(* Logix 5000 project; controller cal1615 1756-L62 rev 20.11; software revision 20.05; part 37 of 82 *)
(* tags used below, declared in another part *)
   FAULT : BOOL;   // Fault AFI
   p01_param_turret_dia_ft : REAL;
   p01r02 : routine;   // System Misc Control
   p01r09_pb_global_reset : BOOL;   // System Modes PB: Global Fault Reset
   p01r12_selected_line_speed : REAL;   // System Line Accel Decel Control Selected Line Speed
   p01r13_line_running : BOOL;   // System Line Start Sequence Line Running
   p01r13_line_slow_ramp : BOOL;   // System Line Start Sequence Start Line to Slow Speed
   p13r03_hz : SYS_SCP;   // Zone 3 Analog Inputs SCP Hz
   p20_acc_fill_time_sec : REAL;   // Letoff Accumulator Fill Time
   p20_acc_input_max : REAL;
   p20_acc_input_min : REAL;
   p20_acc_output_max : REAL;
   p20_acc_output_min : REAL;
   p20_ai_acc_pstn : REAL;   // Letoff Analog Input Accumulator Position
   p20_ai_lc01 : REAL;   // Letoff Analog Input Line Tension Load Cell Splicer
   p20_ai_letoff_dia : REAL;   // Letoff Analog Inputs Letoff Roll Diameter [in]
   p20_ai_lo_turret_amps : REAL;   // Letoff Inputs Letoff Turret VFD Amps
   p20_ai_lo_turret_hz : REAL;   // Letoff Inputs Letoff Turret VFD Hz
   p20_ai_lo_turret_speed : REAL;
   p20_ai_loa_speed : REAL;   // Letoff Inputs Letoff A VFD Surface Speed
   p20_ai_lob_speed : REAL;   // Letoff Inputs Letoff A Speed
   p20_di_acc_door_open : BOOL;
   p20_di_acc_empty : BOOL;   // Letoff Digital Input Letoff Accumulator Empty Position
   p20_di_acc_full : BOOL;   // Letoff Digital Input Letoff Accumulator Full Control Position
   p20_di_clutch_prs_ok : BOOL;   // Letoff Modes Accumulator Position Mode
   p20_di_lfr_jog_fwd : BOOL;   // Letoff Digital Input PB: Feedroll Jog Forward
   p20_di_lfr_jog_rev : BOOL;   // Letoff Digital Input PB: Feedroll Jog Reverse
   p20_di_lfr_nip_close : BOOL;   // Letoff Digital Input PB: Feedroll Nip Roll Close
   p20_di_lo_turret : acs800_di_normal;   // Letoff Letoff Turret VFD Drive Inputs
   p20_di_lo_turret_therm : BOOL;   // Letoff Input Letoff Turret Motor Temp Ok
   p20_di_loa_active : BOOL;   // Letoff Digital Input Letoff A Active
   p20_di_loa_brake : BOOL;   // Letoff Input Letoff A Brake Temperature Ok
   p20_di_loa_fwd_dir : BOOL;   // Letoff Digital Inputs PB: Letoff A Jog FWD
   p20_di_loa_jog : BOOL;   // Letoff Digital Inputs PB: Letoff A Jog REV
   p20_di_loa_start : BOOL;   // Letoff Digital Input PB: Letoff A Start
   p20_di_loa_stop : BOOL;   // Letoff Digital Input PB: Letoff A Stop Stop = 0
   p20_di_loa_temp : BOOL;   // Letoff Input Letoff A Motor Temperature Ok
   p20_di_lob_brake_thermostat : BOOL;   // Letoff Input Letoff B Brake Temperature OK
   p20_di_lob_fwd_dir : BOOL;   // Letoff Digital Inputs PB: Letoff B Jog FWD
   p20_di_lob_jog : BOOL;   // Letoff Digital Inputs PB: Letoff B Jog REV
   p20_di_lob_motor_thermostat : BOOL;   // Letoff Input Letoff B Motor Temperature Ok
   p20_di_lob_start : BOOL;   // Letoff Digital Input PB: Letoff B Start
   p20_di_lob_stop : BOOL;   // Letoff Digital Input PB: Letoff B Stop
   p20_di_lof_acc_fill : BOOL;   // Letoff Digital Input PB: Accumulator Fill
   p20_di_turret_fwd : BOOL;   // Letoff Digital Inputs PB: Turret FWD
   p20_di_turret_pos : BOOL;   // Letoff Digital Inputs PX: Turret in Position
   p20_di_turret_rev : BOOL;   // Letoff Digital Inputs PB: Turret REV
   p20_dia_input_max : REAL;
   p20_dia_input_min : REAL;
   p20_dia_output_max : REAL;
   p20_dia_output_min : REAL;
   p20_dint_to_hmi : DINT[16];   // Letoff Dint to HMI
   p20_lc_input_max : REAL;
   p20_lc_input_min : REAL;   // Letoff Analog Input
   p20_lc_output_max : REAL;
   p20_lc_output_min : REAL;
   p20_loa_ai_amps : REAL;   // Letoff Inputs Letoff A VFD Amps
   p20_loa_ai_hz : REAL;   // Letoff Inputs Letoff A Hz
   p20_loa_ai_rpm : REAL;
   p20_loa_ai_torque : REAL;
   p20_loa_footage_input_max : REAL;
   p20_loa_footage_input_min : REAL;
   p20_loa_footage_output_max : REAL;
   p20_loa_footage_output_min : REAL;
   p20_lob_ai_amps : REAL;   // Letoff Inputs Letoff B VFD Amps
   p20_lob_ai_hz : REAL;   // Letoff Inputs Letoff B VFD Hz
   p20_lob_ai_rpm : REAL;
   p20_lob_ai_torque : REAL;
   p20_lob_footage_input_max : REAL;
   p20_lob_footage_input_min : REAL;
   p20_lob_footage_output_max : REAL;
   p20_lob_footage_output_min : REAL;
   p20_param_lo_turret_gear_ratio : REAL;
   p20_param_loa_gear_ratio : REAL;
   p20_param_lob_gear_ratio : REAL;
   p20_vfd_di_loa : acs800_di_normal;   // Letoff A VFD Inputs
   p20_vfd_di_lob : acs800_di_normal;   // Letoff B VFD Inputs
   p20r01 : routine;   // Letoff Main
   p20r02 : routine;   // Letoff Misc Control
   p20r02_fault_exists : BOOL;
   p20r02_letoff_dia_ft : REAL;   // Letoff Misc Control Letoff Diameter [ft]
   p20r02_letoff_selection_dwell : TIMER;
   p20r02_timer_fault : TIMER[4];   // Letoff Misc Control Fault Delay
   p20r02_timer_warning : TIMER[4];   // Letoff Misc Control Warning Delay
   p20r02_unack_fault : BOOL;   // Letoff Misc Control Unacknowledge Fault Exists
   p20r02_unack_warning : BOOL;   // Letoff Misc Control Unacknowledge Warning Exists
   p20r02_warning_exists : BOOL;
   p20r03 : routine;   // Letoff Input
   p20r03_accumulator_pct_scp : SYS_SCP;   // Letoff Analog Inputs Accumulator Position 0-100%
   p20r03_accumulator_scp : SYS_SCP;   // Letoff Analog Inputs Accumulator Position 0-63 in
   p20r03_distance_to_core : REAL;
   p20r03_lo_radius : REAL;   // Letoff Analog Inputs Letoff Roll Radius
   p20r03_lo_turret_speed_fb : SYS_RPM_TO_SPEED;   // Letoff Inputs Letoff Turret Speed Feedback
   p20r03_loa_distance_to_core : REAL;
   p20r03_Loa_footage_scp : SYS_SCP;   // Letoff Analog Inputs Letoff A Footage Counter Scaling
   p20r03_loa_speed_fb : SYS_RPM_TO_SPEED;   // Letoff Inputs Letoff A VFD Speed Feedback SCP
   p20r03_load_cell : SYS_SCP;   // Letoff Analog Input Load Cell Scaling 0-(2*150lbs)
   p20r03_lob_distance_to_core : REAL;
   p20r03_Lob_footage_scp : SYS_SCP;   // Letoff Analog Inputs Letoff B Footage Counter Scaling
   p20r03_lob_speed_fb : SYS_RPM_TO_SPEED;   // Letoff Inputs Letoff B VFD Speed Feedback SCP
   p20r03_sensor_input : REAL;
   p20r03_sensor_scp : SYS_SCP;   // Letoff Analog Input Sensor Scaling
   p20r03_timer_fault : TIMER[4];   // Letoff Input Fault Delay
   p20r03_timer_warning : TIMER[4];   // Letoff Input Warning Delay
   p20r04 : routine;   // Letoff Ouput
   p20r05 : routine;   // Letoff Dint to HMI
   p20r06 : routine;   // Letoff Real to HMI
   p20r07 : routine;   // Letoff Alarms
   p20r08 : routine;   // Letoff Warnings
   p20r09 : routine;   // Letoff Modes
   p20r10 : routine;   // Letoff Letoff Tension Control
   p20r11 : routine;   // Letoff Feedroll
   p20r13 : routine;   // Letoff Accum Control
   p20r13_ai_acc_pct : REAL;   // Letoff Accumulator Pct Full
   p20r13_ai_loa_footage_ft : REAL;
   p20r13_ai_lob_footage_ft : REAL;
   p20r14 : routine;   // Letoff Accumulator Fill Pressure
   p20r15 : routine;   // Letoff Letoff A VFD
   p20r15_loa_on : BOOL;   // Letoff Letoff A VFD On
   p20r16 : routine;   // Letoff Letoff B VFD
   p20r16_lob_on : BOOL;   // Letoff Letoff B On
   p20r17 : routine;   // Letoff Letoff Diameter Calc
   p20r17_letoff_avg_diam_inch : REAL;   // Letoff Letoff Diameter Calc Average Diameter [in]
   p20r18 : routine;   // Letoff Letoff Turret VFD
   p22_ao_selected_speed : REAL;   // Tension Stand 1 VFD Selected Speed

PROGRAM P20_Letoff   (* main routine R01_Main *)

ROUTINE R01_Main   (* ladder *)
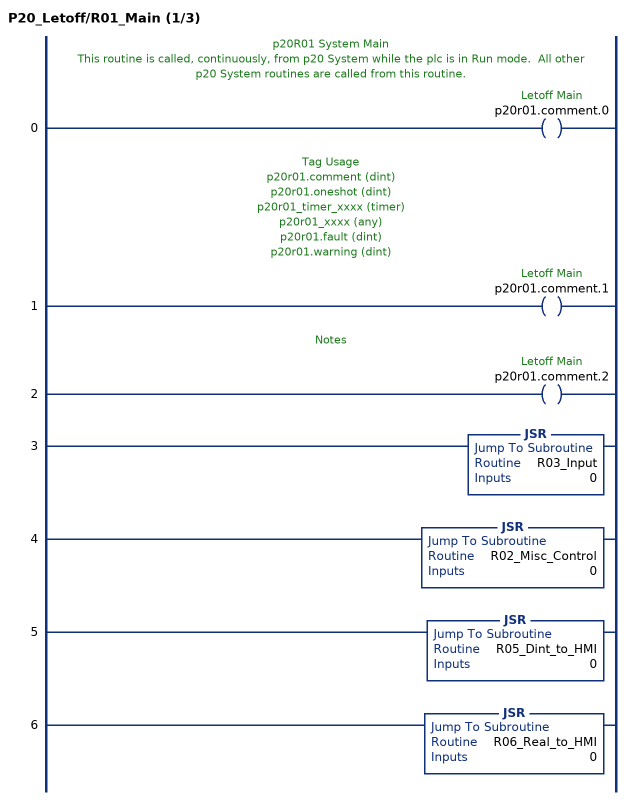
   // p20R01 System Main
   // This routine is called, continuously, from p20 System while the plc is in Run mode.  All other p20 System routines are called from this routine.
   0: OTE(p20r01.comment.0);
   // Tag Usage
   // p20r01.comment (dint)
   // p20r01.oneshot (dint)
   // p20r01_timer_xxxx (timer)
   // p20r01_xxxx (any)
   // p20r01.fault (dint)
   // p20r01.warning (dint)
   1: OTE(p20r01.comment.1);
   // Notes
   2: OTE(p20r01.comment.2);
   3: JSR(R03_Input,0);
   4: JSR(R02_Misc_Control,0);
   5: JSR(R05_Dint_to_HMI,0);
   6: JSR(R06_Real_to_HMI,0);
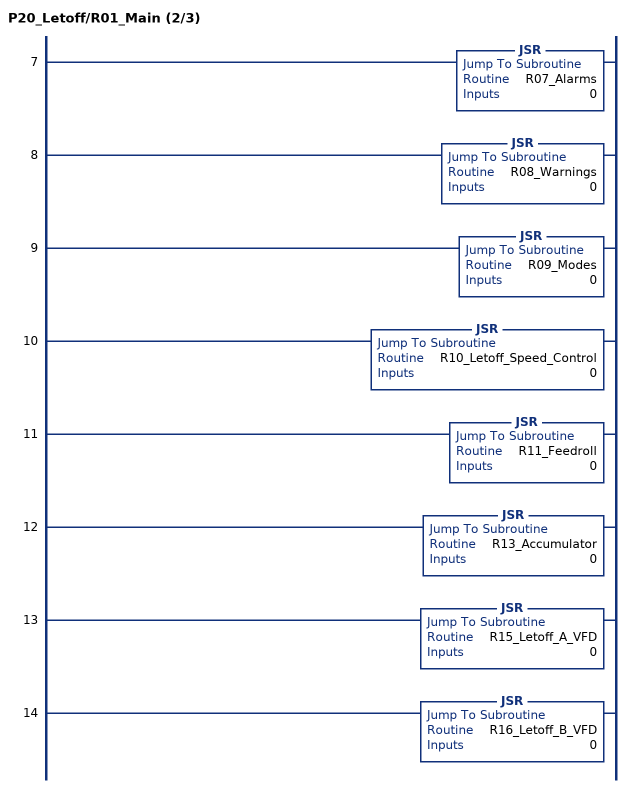
   7: JSR(R07_Alarms,0);
   8: JSR(R08_Warnings,0);
   9: JSR(R09_Modes,0);
   10: JSR(R10_Letoff_Speed_Control,0);
   11: JSR(R11_Feedroll,0);
   12: JSR(R13_Accumulator,0);
   13: JSR(R15_Letoff_A_VFD,0);
   14: JSR(R16_Letoff_B_VFD,0);
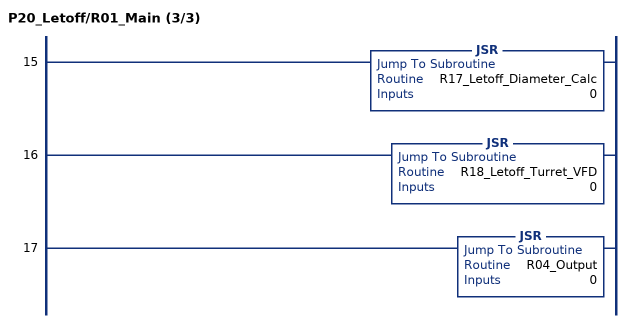
   15: JSR(R17_Letoff_Diameter_Calc,0);
   16: JSR(R18_Letoff_Turret_VFD,0);
   17: JSR(R04_Output,0);
END_ROUTINE

ROUTINE R02_Misc_Control   (* ladder *)
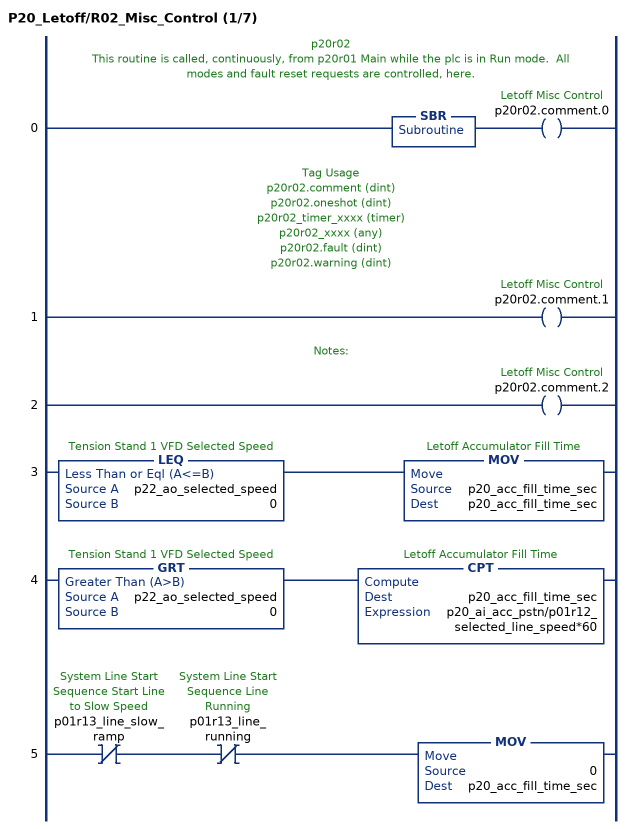
   // p20r02
   // This routine is called, continuously, from p20r01 Main while the plc is in Run mode.  All modes and fault reset requests are controlled, here.
   0: SBR()OTE(p20r02.comment.0);
   // Tag Usage
   // p20r02.comment (dint)
   // p20r02.oneshot (dint)
   // p20r02_timer_xxxx (timer)
   // p20r02_xxxx (any)
   // p20r02.fault (dint)
   // p20r02.warning (dint)
   1: OTE(p20r02.comment.1);
   // Notes:
   2: OTE(p20r02.comment.2);
   3: LEQ(p22_ao_selected_speed,0)MOV(p20_acc_fill_time_sec,p20_acc_fill_time_sec);
   4: GRT(p22_ao_selected_speed,0)CPT(p20_acc_fill_time_sec,p20_ai_acc_pstn/p01r12_selected_line_speed*60);
   5: XIO(p01r13_line_slow_ramp)XIO(p01r13_line_running)MOV(0,p20_acc_fill_time_sec);
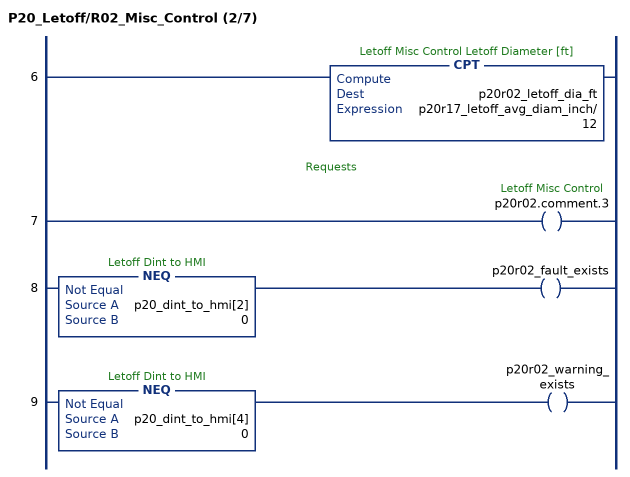
   6: CPT(p20r02_letoff_dia_ft,p20r17_letoff_avg_diam_inch/12);
   // Requests
   7: OTE(p20r02.comment.3);
   8: NEQ(p20_dint_to_hmi[2],0)OTE(p20r02_fault_exists);
   9: NEQ(p20_dint_to_hmi[4],0)OTE(p20r02_warning_exists);
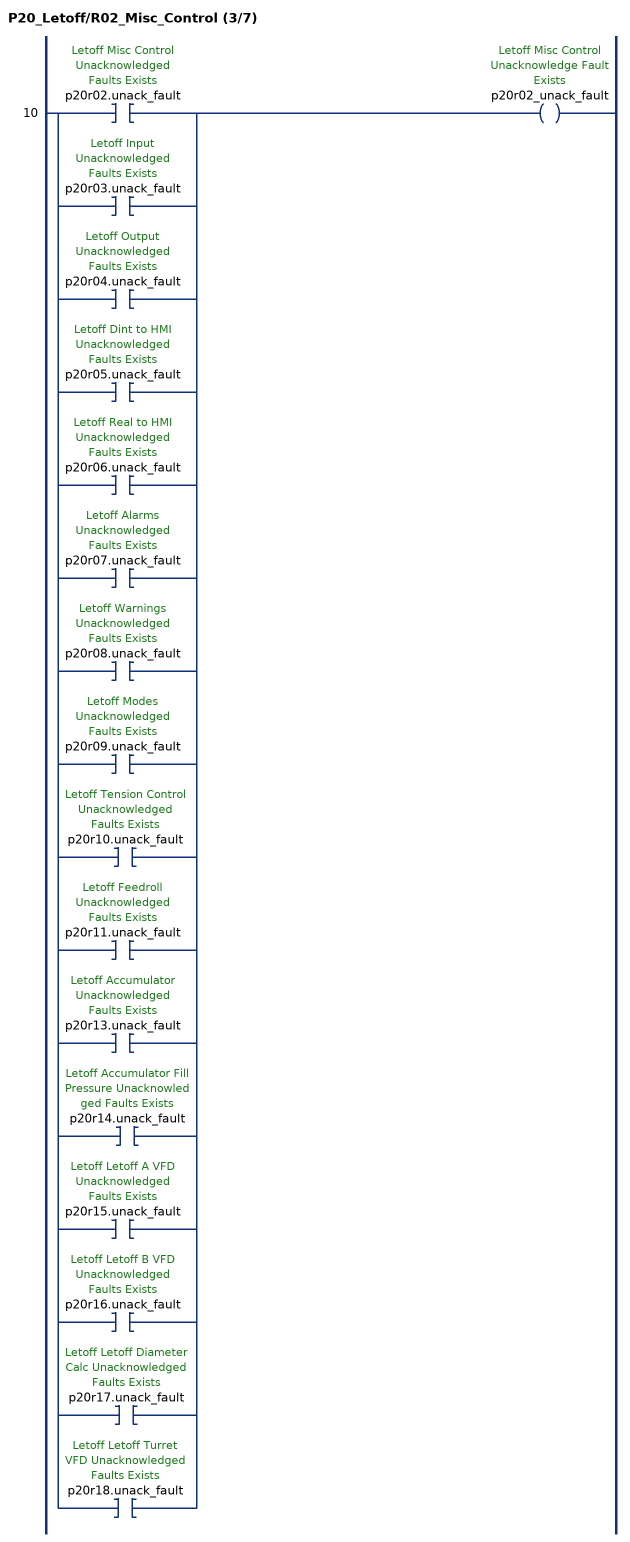
   10: [XIC(p20r02.unack_fault) ,XIC(p20r03.unack_fault) ,XIC(p20r04.unack_fault) ,XIC(p20r05.unack_fault) ,XIC(p20r06.unack_fault) ,XIC(p20r07.unack_fault) ,XIC(p20r08.unack_fault) ,XIC(p20r09.unack_fault) ,XIC(p20r10.unack_fault) ,XIC(p20r11.unack_fault) ,XIC(p20r13.unack_fault) ,XIC(p20r14.unack_fault) ,XIC(p20r15.unack_fault) ,XIC(p20r16.unack_fault) ,XIC(p20r17.unack_fault) ,XIC(p20r18.unack_fault) ]OTE(p20r02_unack_fault);
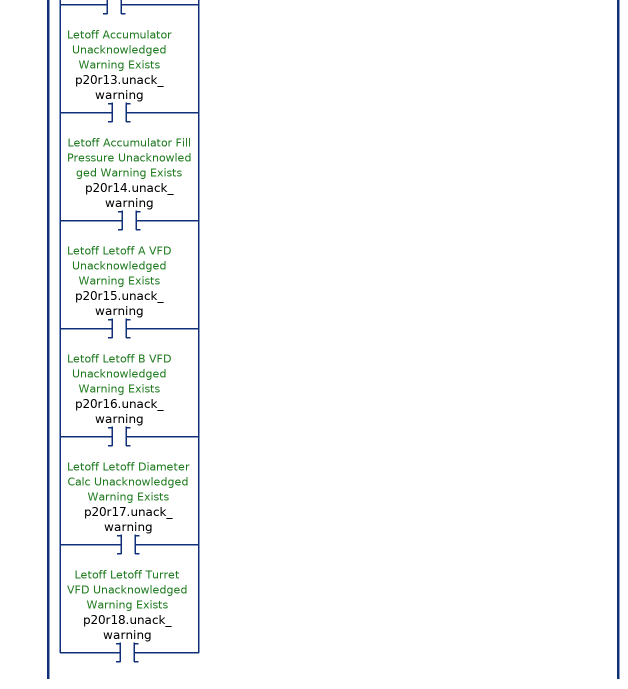
   11: [XIC(p20r02.unack_warning) ,XIC(p20r03.unack_warning) ,XIC(p20r04.unack_warning) ,XIC(p20r05.unack_warning) ,XIC(p20r06.unack_warning) ,XIC(p20r07.unack_warning) ,XIC(p20r08.unack_warning) ,XIC(p20r09.unack_warning) ,XIC(p20r10.unack_warning) ,XIC(p20r11.unack_warning) ,XIC(p20r13.unack_warning) ,XIC(p20r14.unack_warning) ,XIC(p20r15.unack_warning) ,XIC(p20r16.unack_warning) ,XIC(p20r17.unack_warning) ,XIC(p20r18.unack_warning) ]OTE(p20r02_unack_warning);
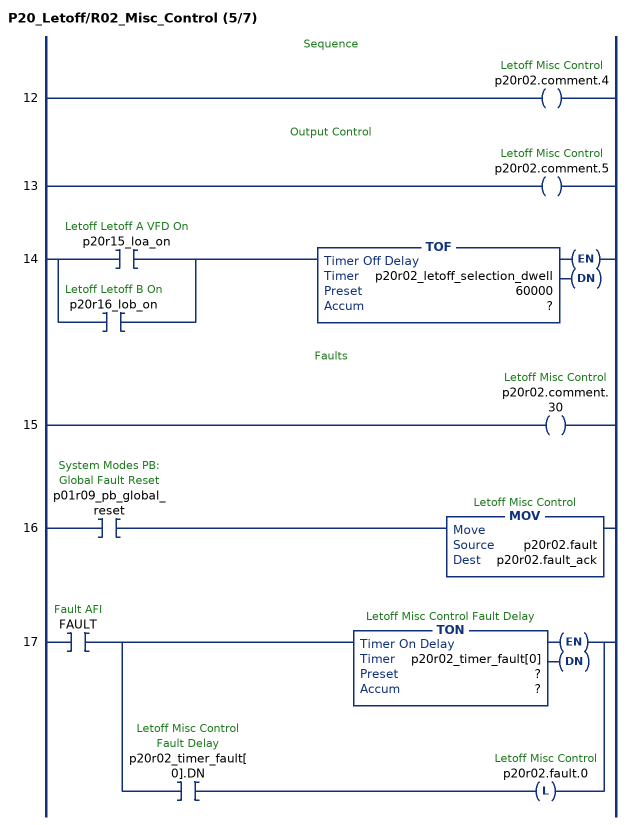
   // Sequence
   12: OTE(p20r02.comment.4);
   // Output Control
   13: OTE(p20r02.comment.5);
   14: [XIC(p20r15_loa_on) ,XIC(p20r16_lob_on) ]TOF(p20r02_letoff_selection_dwell,?,?);
   // Faults
   15: OTE(p20r02.comment.30);
   16: XIC(p01r09_pb_global_reset)MOV(p20r02.fault,p20r02.fault_ack);
   17: XIC(FAULT)[TON(p20r02_timer_fault[0],?,?) ,XIC(p20r02_timer_fault[0].DN) OTL(p20r02.fault.0) ];
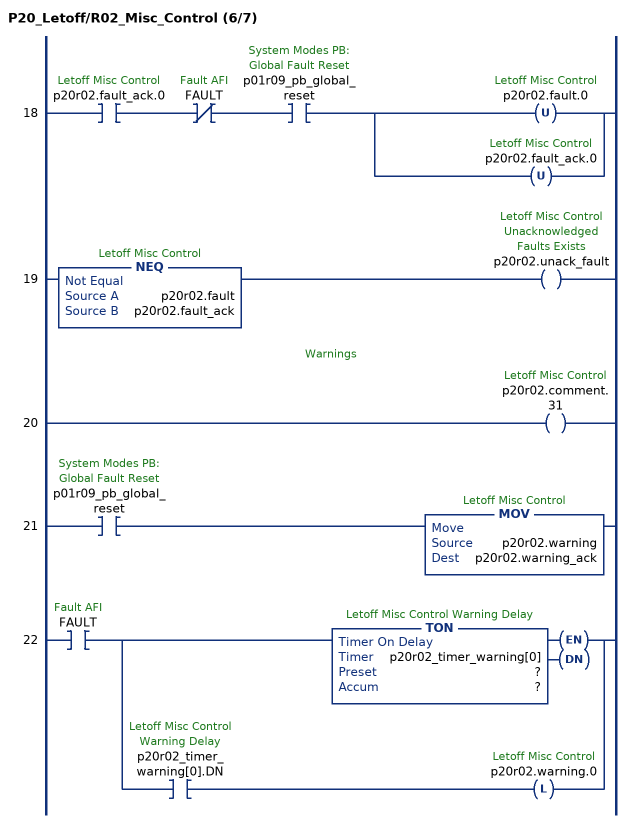
   18: XIC(p20r02.fault_ack.0)XIO(FAULT)XIC(p01r09_pb_global_reset)[OTU(p20r02.fault.0) ,OTU(p20r02.fault_ack.0) ];
   19: NEQ(p20r02.fault,p20r02.fault_ack)OTE(p20r02.unack_fault);
   // Warnings
   20: OTE(p20r02.comment.31);
   21: XIC(p01r09_pb_global_reset)MOV(p20r02.warning,p20r02.warning_ack);
   22: XIC(FAULT)[TON(p20r02_timer_warning[0],?,?) ,XIC(p20r02_timer_warning[0].DN) OTL(p20r02.warning.0) ];
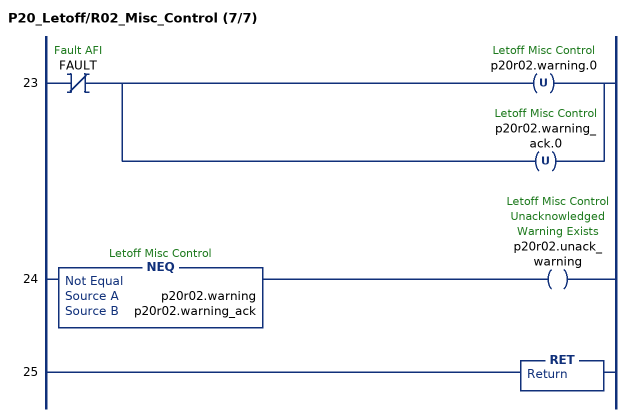
   23: XIO(FAULT)[OTU(p20r02.warning.0) ,OTU(p20r02.warning_ack.0) ];
   24: NEQ(p20r02.warning,p20r02.warning_ack)OTE(p20r02.unack_warning);
   25: RET();
END_ROUTINE

ROUTINE R03_Input   (* ladder *)
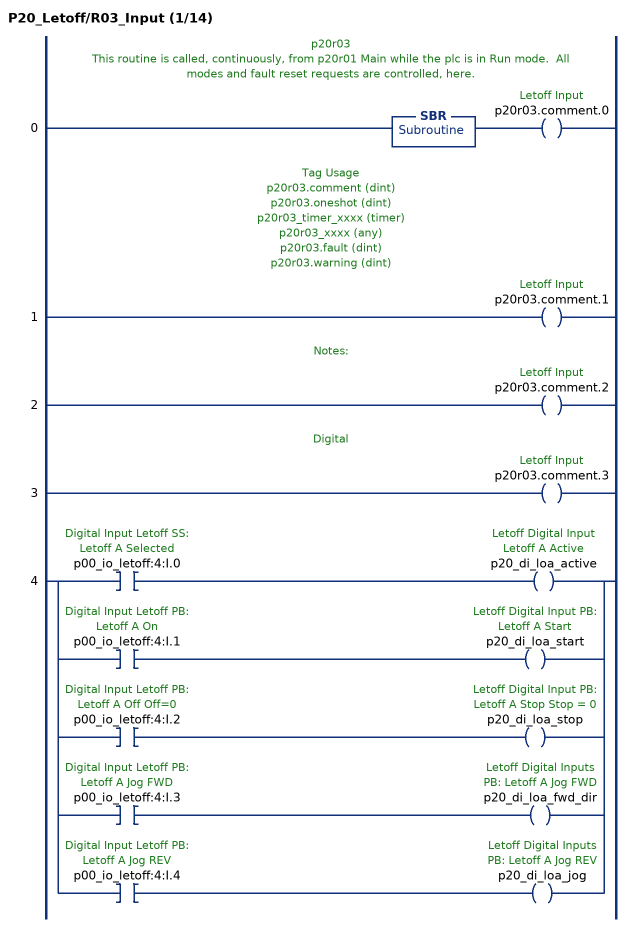
   // p20r03
   // This routine is called, continuously, from p20r01 Main while the plc is in Run mode.  All modes and fault reset requests are controlled, here.
   0: SBR()OTE(p20r03.comment.0);
   // Tag Usage
   // p20r03.comment (dint)
   // p20r03.oneshot (dint)
   // p20r03_timer_xxxx (timer)
   // p20r03_xxxx (any)
   // p20r03.fault (dint)
   // p20r03.warning (dint)
   1: OTE(p20r03.comment.1);
   // Notes:
   2: OTE(p20r03.comment.2);
   // Digital
   3: OTE(p20r03.comment.3);
   4: [XIC(p00_io_letoff:4:I.0) OTE(p20_di_loa_active) ,XIC(p00_io_letoff:4:I.1) OTE(p20_di_loa_start) ,XIC(p00_io_letoff:4:I.2) OTE(p20_di_loa_stop) ,XIC(p00_io_letoff:4:I.3) OTE(p20_di_loa_fwd_dir) ,XIC(p00_io_letoff:4:I.4) OTE(p20_di_loa_jog) ];
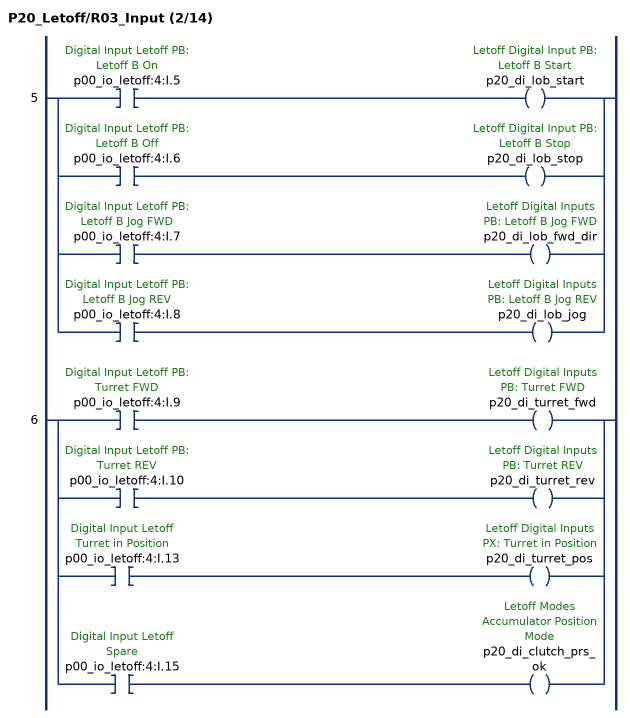
   5: [XIC(p00_io_letoff:4:I.5) OTE(p20_di_lob_start) ,XIC(p00_io_letoff:4:I.6) OTE(p20_di_lob_stop) ,XIC(p00_io_letoff:4:I.7) OTE(p20_di_lob_fwd_dir) ,XIC(p00_io_letoff:4:I.8) OTE(p20_di_lob_jog) ];
   6: [XIC(p00_io_letoff:4:I.9) OTE(p20_di_turret_fwd) ,XIC(p00_io_letoff:4:I.10) OTE(p20_di_turret_rev) ,XIC(p00_io_letoff:4:I.13) OTE(p20_di_turret_pos) ,XIC(p00_io_letoff:4:I.15) OTE(p20_di_clutch_prs_ok) ];
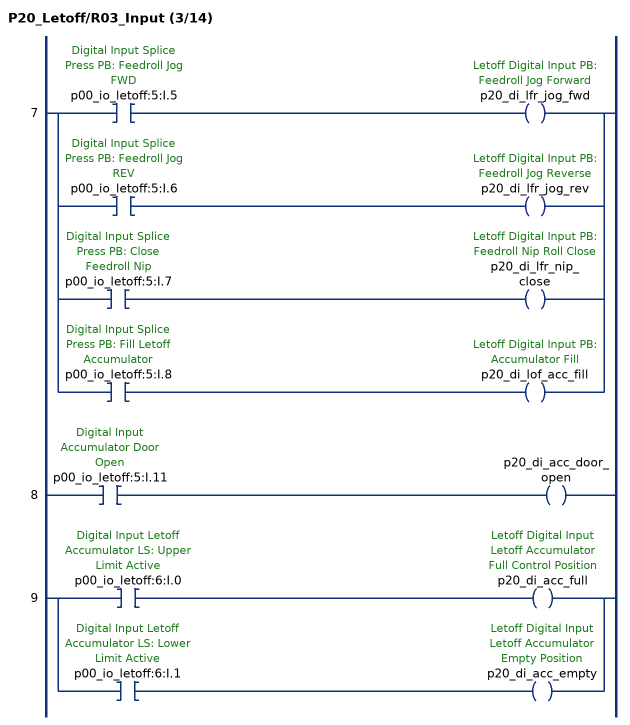
   7: [XIC(p00_io_letoff:5:I.5) OTE(p20_di_lfr_jog_fwd) ,XIC(p00_io_letoff:5:I.6) OTE(p20_di_lfr_jog_rev) ,XIC(p00_io_letoff:5:I.7) OTE(p20_di_lfr_nip_close) ,XIC(p00_io_letoff:5:I.8) OTE(p20_di_lof_acc_fill) ];
   8: XIC(p00_io_letoff:5:I.11)OTE(p20_di_acc_door_open);
   9: [XIC(p00_io_letoff:6:I.0) OTE(p20_di_acc_full) ,XIC(p00_io_letoff:6:I.1) OTE(p20_di_acc_empty) ];
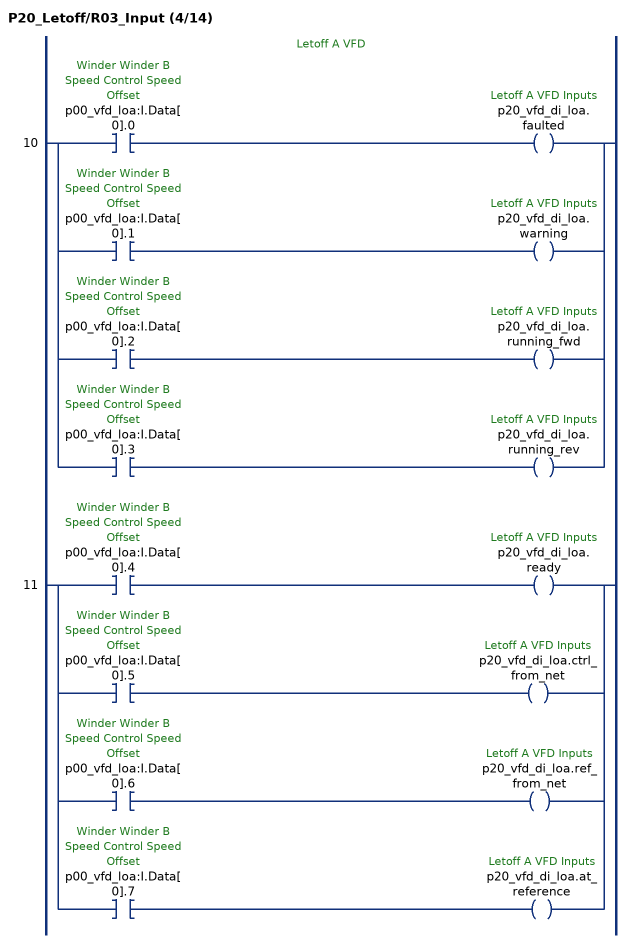
   // Letoff A VFD
   10: [XIC(p00_vfd_loa:I.Data[0].0) OTE(p20_vfd_di_loa.faulted) ,XIC(p00_vfd_loa:I.Data[0].1) OTE(p20_vfd_di_loa.warning) ,XIC(p00_vfd_loa:I.Data[0].2) OTE(p20_vfd_di_loa.running_fwd) ,XIC(p00_vfd_loa:I.Data[0].3) OTE(p20_vfd_di_loa.running_rev) ];
   11: [XIC(p00_vfd_loa:I.Data[0].4) OTE(p20_vfd_di_loa.ready) ,XIC(p00_vfd_loa:I.Data[0].5) OTE(p20_vfd_di_loa.ctrl_from_net) ,XIC(p00_vfd_loa:I.Data[0].6) OTE(p20_vfd_di_loa.ref_from_net) ,XIC(p00_vfd_loa:I.Data[0].7) OTE(p20_vfd_di_loa.at_reference) ];
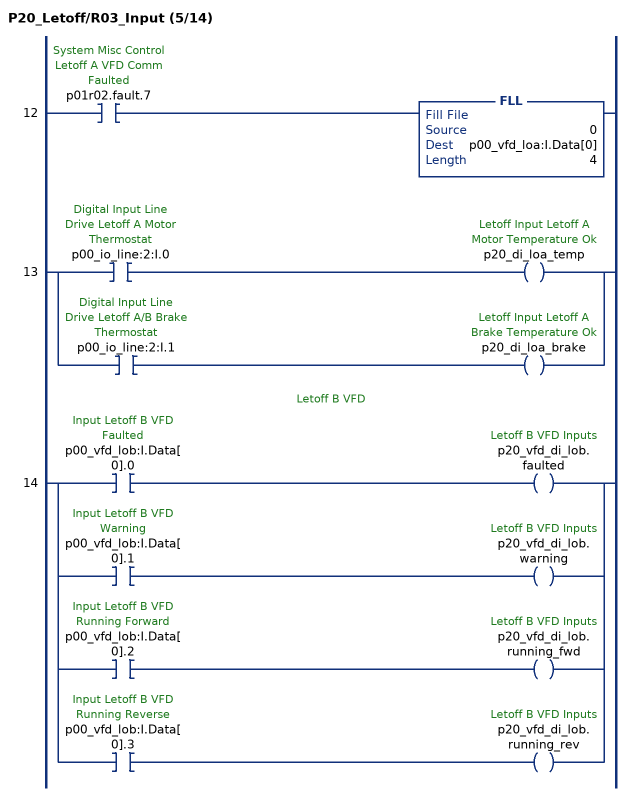
   12: XIC(p01r02.fault.7)FLL(0,p00_vfd_loa:I.Data[0],4);
   13: [XIC(p00_io_line:2:I.0) OTE(p20_di_loa_temp) ,XIC(p00_io_line:2:I.1) OTE(p20_di_loa_brake) ];
   // Letoff B VFD
   14: [XIC(p00_vfd_lob:I.Data[0].0) OTE(p20_vfd_di_lob.faulted) ,XIC(p00_vfd_lob:I.Data[0].1) OTE(p20_vfd_di_lob.warning) ,XIC(p00_vfd_lob:I.Data[0].2) OTE(p20_vfd_di_lob.running_fwd) ,XIC(p00_vfd_lob:I.Data[0].3) OTE(p20_vfd_di_lob.running_rev) ];
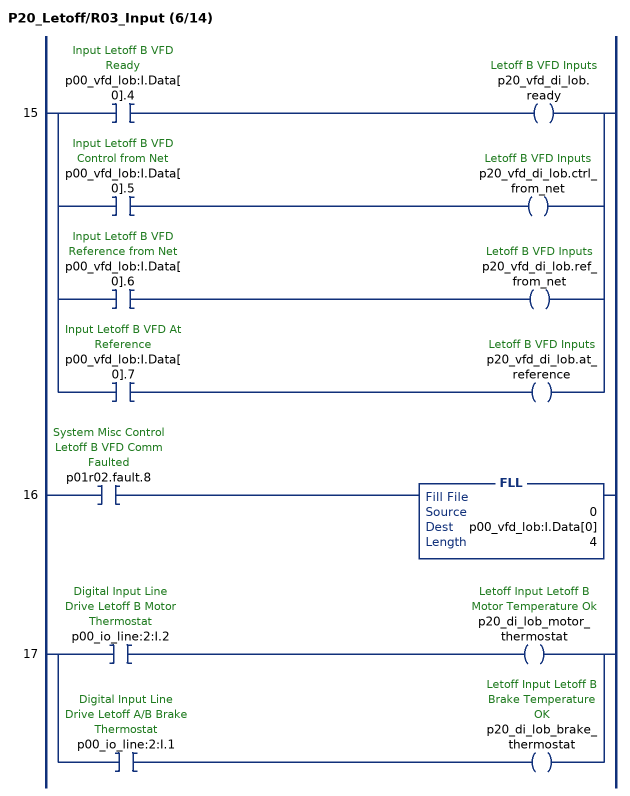
   15: [XIC(p00_vfd_lob:I.Data[0].4) OTE(p20_vfd_di_lob.ready) ,XIC(p00_vfd_lob:I.Data[0].5) OTE(p20_vfd_di_lob.ctrl_from_net) ,XIC(p00_vfd_lob:I.Data[0].6) OTE(p20_vfd_di_lob.ref_from_net) ,XIC(p00_vfd_lob:I.Data[0].7) OTE(p20_vfd_di_lob.at_reference) ];
   16: XIC(p01r02.fault.8)FLL(0,p00_vfd_lob:I.Data[0],4);
   17: [XIC(p00_io_line:2:I.2) OTE(p20_di_lob_motor_thermostat) ,XIC(p00_io_line:2:I.1) OTE(p20_di_lob_brake_thermostat) ];
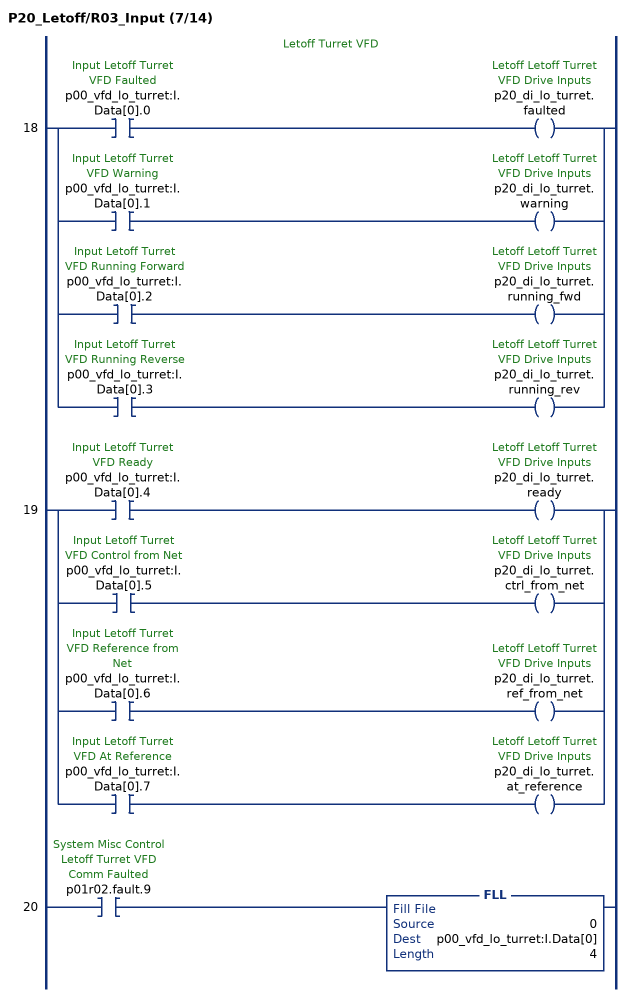
   // Letoff Turret VFD
   18: [XIC(p00_vfd_lo_turret:I.Data[0].0) OTE(p20_di_lo_turret.faulted) ,XIC(p00_vfd_lo_turret:I.Data[0].1) OTE(p20_di_lo_turret.warning) ,XIC(p00_vfd_lo_turret:I.Data[0].2) OTE(p20_di_lo_turret.running_fwd) ,XIC(p00_vfd_lo_turret:I.Data[0].3) OTE(p20_di_lo_turret.running_rev) ];
   19: [XIC(p00_vfd_lo_turret:I.Data[0].4) OTE(p20_di_lo_turret.ready) ,XIC(p00_vfd_lo_turret:I.Data[0].5) OTE(p20_di_lo_turret.ctrl_from_net) ,XIC(p00_vfd_lo_turret:I.Data[0].6) OTE(p20_di_lo_turret.ref_from_net) ,XIC(p00_vfd_lo_turret:I.Data[0].7) OTE(p20_di_lo_turret.at_reference) ];
   20: XIC(p01r02.fault.9)FLL(0,p00_vfd_lo_turret:I.Data[0],4);
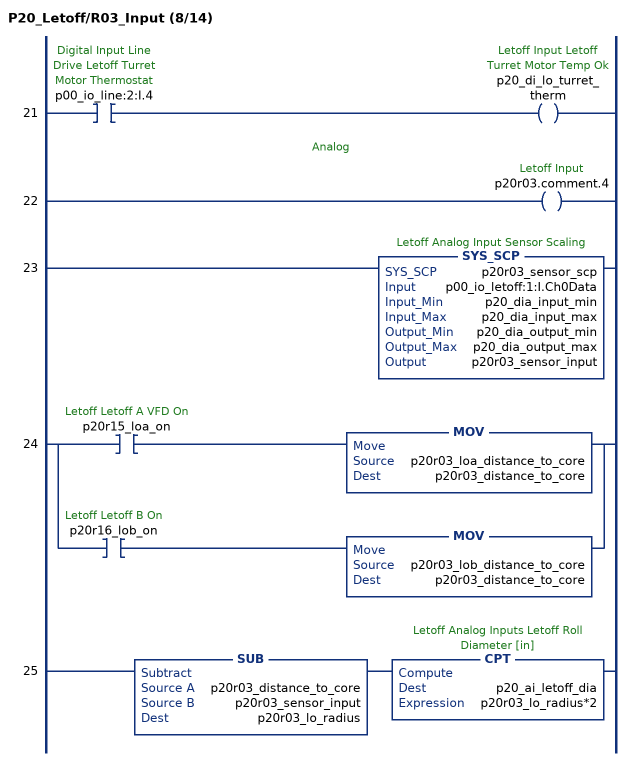
   21: XIC(p00_io_line:2:I.4)OTE(p20_di_lo_turret_therm);
   // Analog
   22: OTE(p20r03.comment.4);
   23: SYS_SCP(p20r03_sensor_scp,p00_io_letoff:1:I.Ch0Data,p20_dia_input_min,p20_dia_input_max,p20_dia_output_min,p20_dia_output_max,p20r03_sensor_input);
   24: [XIC(p20r15_loa_on) MOV(p20r03_loa_distance_to_core,p20r03_distance_to_core) ,XIC(p20r16_lob_on) MOV(p20r03_lob_distance_to_core,p20r03_distance_to_core) ];
   25: SUB(p20r03_distance_to_core,p20r03_sensor_input,p20r03_lo_radius)CPT(p20_ai_letoff_dia,p20r03_lo_radius*2);
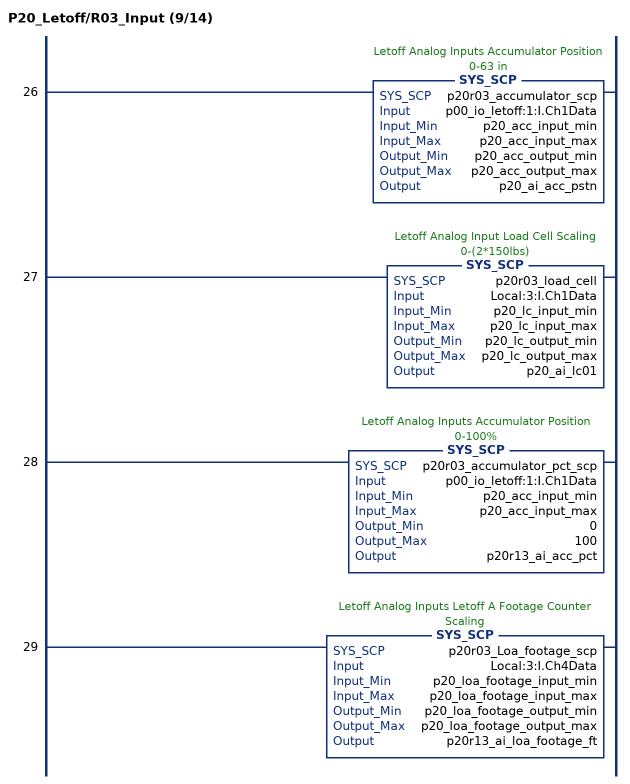
   26: SYS_SCP(p20r03_accumulator_scp,p00_io_letoff:1:I.Ch1Data,p20_acc_input_min,p20_acc_input_max,p20_acc_output_min,p20_acc_output_max,p20_ai_acc_pstn);
   27: SYS_SCP(p20r03_load_cell,Local:3:I.Ch1Data,p20_lc_input_min,p20_lc_input_max,p20_lc_output_min,p20_lc_output_max,p20_ai_lc01);
   28: SYS_SCP(p20r03_accumulator_pct_scp,p00_io_letoff:1:I.Ch1Data,p20_acc_input_min,p20_acc_input_max,0,100,p20r13_ai_acc_pct);
   29: SYS_SCP(p20r03_Loa_footage_scp,Local:3:I.Ch4Data,p20_loa_footage_input_min,p20_loa_footage_input_max,p20_loa_footage_output_min,p20_loa_footage_output_max,p20r13_ai_loa_footage_ft);
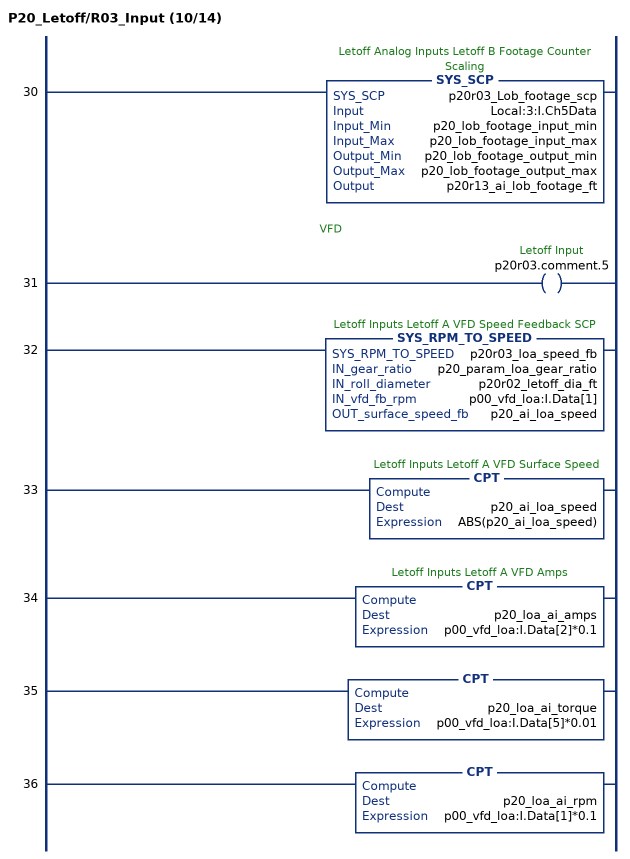
   30: SYS_SCP(p20r03_Lob_footage_scp,Local:3:I.Ch5Data,p20_lob_footage_input_min,p20_lob_footage_input_max,p20_lob_footage_output_min,p20_lob_footage_output_max,p20r13_ai_lob_footage_ft);
   // VFD
   31: OTE(p20r03.comment.5);
   32: SYS_RPM_TO_SPEED(p20r03_loa_speed_fb,p20_param_loa_gear_ratio,p20r02_letoff_dia_ft,p00_vfd_loa:I.Data[1],p20_ai_loa_speed);
   33: CPT(p20_ai_loa_speed,ABS(p20_ai_loa_speed));
   34: CPT(p20_loa_ai_amps,p00_vfd_loa:I.Data[2]*0.1);
   35: CPT(p20_loa_ai_torque,p00_vfd_loa:I.Data[5]*0.01);
   36: CPT(p20_loa_ai_rpm,p00_vfd_loa:I.Data[1]*0.1);
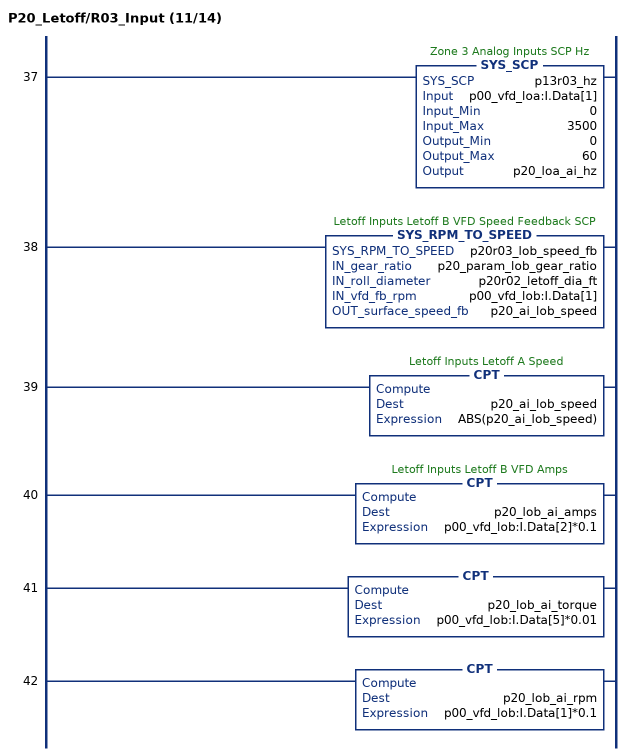
   37: SYS_SCP(p13r03_hz,p00_vfd_loa:I.Data[1],0,3500,0,60,p20_loa_ai_hz);
   38: SYS_RPM_TO_SPEED(p20r03_lob_speed_fb,p20_param_lob_gear_ratio,p20r02_letoff_dia_ft,p00_vfd_lob:I.Data[1],p20_ai_lob_speed);
   39: CPT(p20_ai_lob_speed,ABS(p20_ai_lob_speed));
   40: CPT(p20_lob_ai_amps,p00_vfd_lob:I.Data[2]*0.1);
   41: CPT(p20_lob_ai_torque,p00_vfd_lob:I.Data[5]*0.01);
   42: CPT(p20_lob_ai_rpm,p00_vfd_lob:I.Data[1]*0.1);
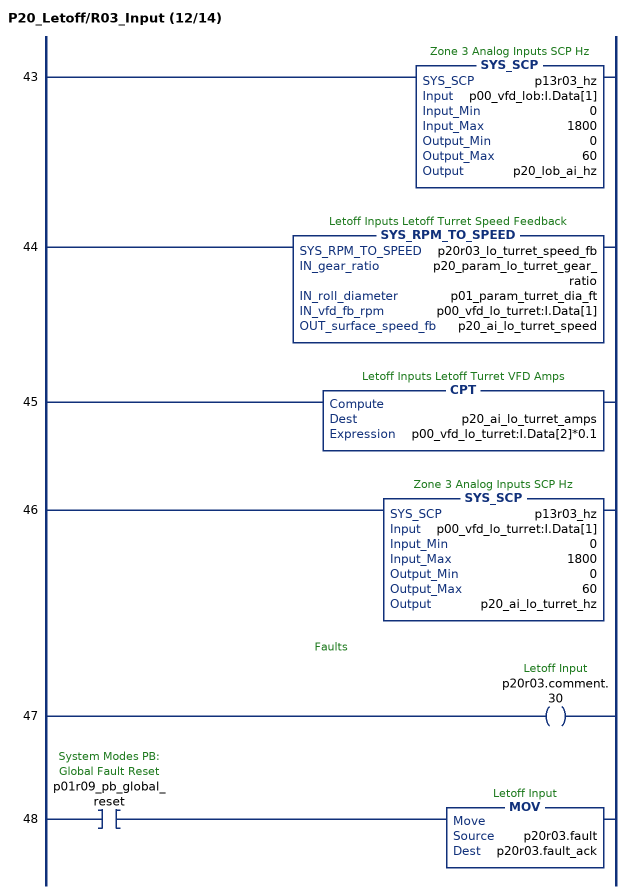
   43: SYS_SCP(p13r03_hz,p00_vfd_lob:I.Data[1],0,1800,0,60,p20_lob_ai_hz);
   44: SYS_RPM_TO_SPEED(p20r03_lo_turret_speed_fb,p20_param_lo_turret_gear_ratio,p01_param_turret_dia_ft,p00_vfd_lo_turret:I.Data[1],p20_ai_lo_turret_speed);
   45: CPT(p20_ai_lo_turret_amps,p00_vfd_lo_turret:I.Data[2]*0.1);
   46: SYS_SCP(p13r03_hz,p00_vfd_lo_turret:I.Data[1],0,1800,0,60,p20_ai_lo_turret_hz);
   // Faults
   47: OTE(p20r03.comment.30);
   48: XIC(p01r09_pb_global_reset)MOV(p20r03.fault,p20r03.fault_ack);
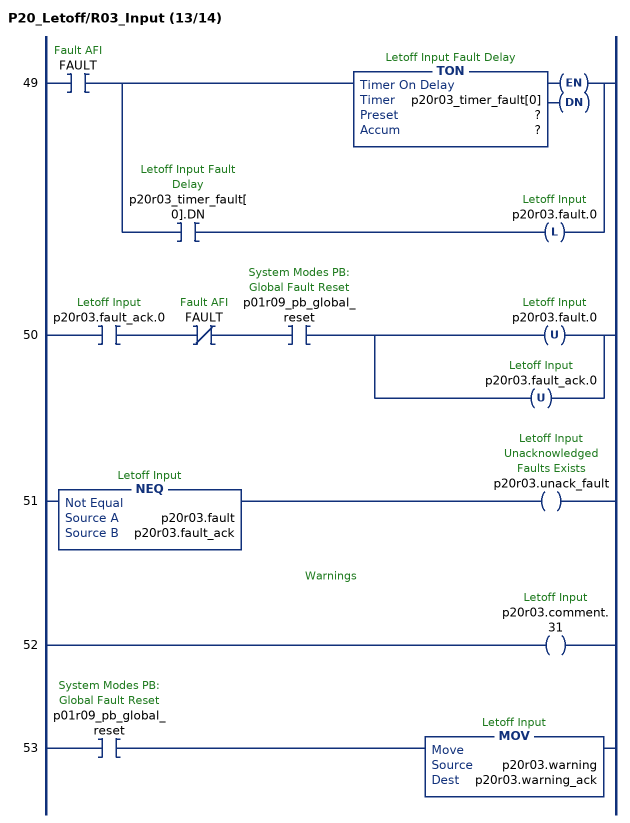
   49: XIC(FAULT)[TON(p20r03_timer_fault[0],?,?) ,XIC(p20r03_timer_fault[0].DN) OTL(p20r03.fault.0) ];
   50: XIC(p20r03.fault_ack.0)XIO(FAULT)XIC(p01r09_pb_global_reset)[OTU(p20r03.fault.0) ,OTU(p20r03.fault_ack.0) ];
   51: NEQ(p20r03.fault,p20r03.fault_ack)OTE(p20r03.unack_fault);
   // Warnings
   52: OTE(p20r03.comment.31);
   53: XIC(p01r09_pb_global_reset)MOV(p20r03.warning,p20r03.warning_ack);
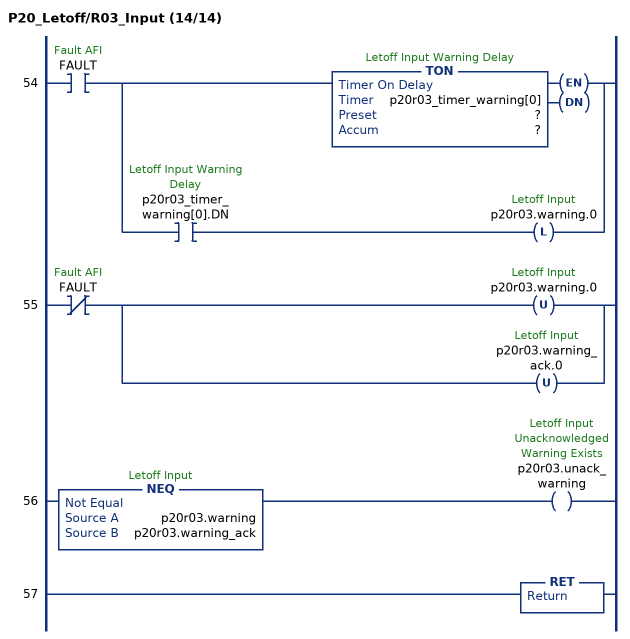
   54: XIC(FAULT)[TON(p20r03_timer_warning[0],?,?) ,XIC(p20r03_timer_warning[0].DN) OTL(p20r03.warning.0) ];
   55: XIO(FAULT)[OTU(p20r03.warning.0) ,OTU(p20r03.warning_ack.0) ];
   56: NEQ(p20r03.warning,p20r03.warning_ack)OTE(p20r03.unack_warning);
   57: RET();
END_ROUTINE
